FUNCTION_BLOCK Utilities_HMI (* Service Interface Function Block Type *)
  (* Standard: 61499-2 *)
  (* Version 0.0, 9/9/2024, SESA685388, Schneider Electric, template *)
  PACKAGE SE.Nereda;
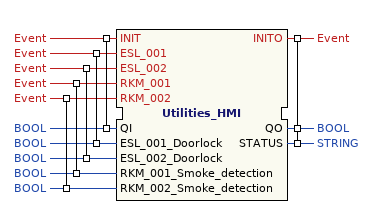
  EVENT_INPUT
    INIT WITH QI;
    ESL_001 WITH ESL_001_Doorlock;
    ESL_002 WITH ESL_002_Doorlock;
    RKM_001 WITH RKM_001_Smoke_detection;
    RKM_002 WITH RKM_002_Smoke_detection;
  END_EVENT
  EVENT_OUTPUT
    INITO WITH QO, STATUS;
  END_EVENT
  VAR_INPUT
    QI : BOOL;
    ESL_001_Doorlock : BOOL;
    ESL_002_Doorlock : BOOL;
    RKM_001_Smoke_detection : BOOL;
    RKM_002_Smoke_detection : BOOL;
  END_VAR
  VAR_OUTPUT
    QO : BOOL; (* Event Output Qualifier *)
    STATUS : STRING; (* Service Status *)
  END_VAR
  SERVICE /
    SEQUENCE 
    END_SEQUENCE
  END_SERVICE
END_FUNCTION_BLOCK
